# B&R Automation Studio project Pors
Automation Studio 4.5.2.102

## Configuration Config1

### Hardware
```
4PP065_0571_P74 : 4PP065.0571-P74 v1.1.2.0
  Connector IF5:
    ActivateDevice = 1
  ConfigurationID = POlaba1_Config1
  Simulation = 1
```

## Logical view

### Library Logical/Libraries/MotContr (ANSIC)

#### MotContr.fun - Exported functions and function blocks
```iecst
{REDUND_ERROR} FUNCTION_BLOCK FB_Integrator (*TODO: Add your comment here*) (*$GROUP=User,$CAT=User,$GROUPICON=User.png,$CATICON=User.png*)
	VAR_INPUT
		in : {REDUND_UNREPLICABLE} REAL;
	END_VAR
	VAR_OUTPUT
		out : {REDUND_UNREPLICABLE} REAL;
	END_VAR
	VAR_INPUT
		dt : REAL;
	END_VAR
	VAR
		prev_value : REAL;
	END_VAR
END_FUNCTION_BLOCK

{REDUND_ERROR} FUNCTION_BLOCK FB_Regulator (*TODO: Add your comment here*) (*$GROUP=User,$CAT=User,$GROUPICON=User.png,$CATICON=User.png*)
	VAR_INPUT
		e_in : {REDUND_UNREPLICABLE} REAL;
	END_VAR
	VAR_OUTPUT
		u_out : {REDUND_UNREPLICABLE} REAL;
	END_VAR
	VAR
		k_p : {REDUND_UNREPLICABLE} REAL;
		k_i : {REDUND_UNREPLICABLE} REAL;
		integrator : {REDUND_UNREPLICABLE} FB_Integrator;
		iyOld : {REDUND_UNREPLICABLE} REAL;
		max_abs_value : {REDUND_UNREPLICABLE} REAL;
	END_VAR
	VAR_INPUT
		dt : REAL;
	END_VAR
	VAR
		last_sum : {REDUND_UNREPLICABLE} REAL;
		sum : {REDUND_UNREPLICABLE} REAL;
	END_VAR
END_FUNCTION_BLOCK

{REDUND_ERROR} FUNCTION_BLOCK FB_Motor (*TODO: Add your comment here*) (*$GROUP=User,$CAT=User,$GROUPICON=User.png,$CATICON=User.png*)
	VAR_INPUT
		u : REAL;
	END_VAR
	VAR_OUTPUT
		w : REAL;
		phi : REAL;
	END_VAR
	VAR
		Tm : REAL;
		integrator : FB_Integrator;
		ke : REAL;
	END_VAR
	VAR_INPUT
		dt : REAL;
	END_VAR
END_FUNCTION_BLOCK
```

### Program Logical/Program (ANSIC)

#### Main.c - Initialization code
```c
#include <bur/plctypes.h>

#ifdef _DEFAULT_INCLUDES
	#include <AsDefault.h>
#endif

void _INIT ProgramInit(void)
{
	fb_motor1.dt = 0.03;
	fb_motor1.ke = 0.30;
	fb_motor1.Tm = 0.1;

	fb_motor2.dt = 0.03;
	fb_motor2.ke = 0.30;
	fb_motor2.Tm = 0.1;

	fb_controller.dt = 0.01;
	fb_controller.k_i = 4.8;
	fb_controller.k_p = 0.48;
	fb_controller.max_abs_value = 24.0;

	speed = 0;
	counter = 0;
	enable = 1;
}
```

#### Cyclic.c - Cyclic code
```c
#include <bur/plctypes.h>

#ifdef _DEFAULT_INCLUDES
	#include <AsDefault.h>
#endif

void _CYCLIC ProgramCyclic(void)
{
	if(enable)
	{
		if(counter == 1000)
		{
			speed = 60;
		}
		if(counter == 1100)
		{
			speed = 0;
			counter = 0;
		}
		counter = counter + 1;

		fb_controller.e_in = speed - fb_motor1.w;
		FB_Regulator(&fb_controller);

		fb_motor1.u = fb_controller.u_out;
		FB_Motor(&fb_motor1);

		fb_motor2.u = speed * fb_motor2.ke;
		FB_Motor(&fb_motor2);

	}
}
```

#### Variables.var - Local variables
```iecst
VAR
	fb_controller : FB_Regulator;
	fb_motor1 : FB_Motor;
	fb_motor2 : FB_Motor;
	speed : REAL;
	counter : UINT;
	enable : {REDUND_UNREPLICABLE} BOOL;
END_VAR
```

Listed in the project but not available here: Logical/Libraries/MotContr/Types.typ, Logical/Libraries/MotContr/Constants.var, Logical/Libraries/MotContr/FB_Regulator.c, Logical/Libraries/MotContr/FB_Motor.c, Logical/Libraries/MotContr/FB_Integrator.c, Logical/Program/Exit.c, Logical/Program/Types.typ
